PROGRAM Vision_1
VAR
	TON_0: TON;
	Always_ON	:	BOOL	:=TRUE	;//상시 ON
	Always_OFF	:	BOOL	:=FALSE	;//상시 OFF

	

    TON_100MS : TON;
    tPreset_Time : TIME := T#100MS;
	bRun_Timer	:	BOOL	;
	
END_VAR

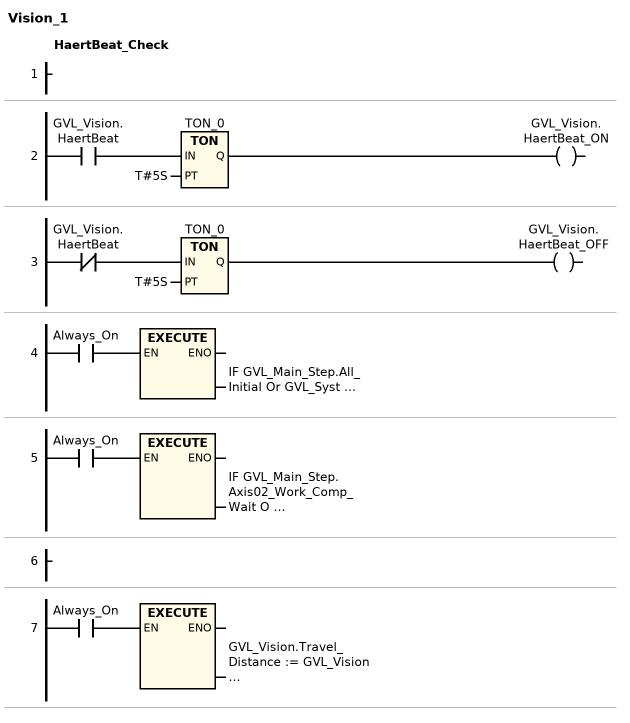
// NETWORK 1: HaertBeat_Check

// NETWORK 2
TON_0(IN := GVL_Vision.HaertBeat, PT := T#5S); // TON
GVL_Vision.HaertBeat_ON := TON_0.Q;

// NETWORK 3
TON_0(IN := NOT GVL_Vision.HaertBeat, PT := T#5S); // TON
GVL_Vision.HaertBeat_OFF := TON_0.Q;

// NETWORK 4
IF Always_On THEN
    IF GVL_Main_Step.All_Initial Or GVL_System.Alarm_Reset THEN
        (* All_Initial이 TRUE일 때, Frame Time을 0으로 초기화 *)
        GVL_Vision.Get_Frame_Time := 0.0;
    END_IF
    bRun_Timer :=GVL_Vision.Vision_Ok AND NOT GVL_Main_Step.Axis04_Work_Comp_Wait;
    TON_100MS(
        IN := bRun_Timer,  
        PT := tPreset_Time,          
        Q  => ,                      
        ET => 
    );
    IF TON_100MS.Q THEN
        
        GVL_Vision.Get_Frame_Time := GVL_Vision.Get_Frame_Time + 0.1;
    	TON_100MS(IN := FALSE);
    
    END_IF
END_IF

// NETWORK 5
IF Always_On THEN
    IF GVL_Main_Step.Axis02_Work_Comp_Wait OR GVL_System.All_Initial THEN
    	GVL_Vision.Data_Read_X	:=	0;
    	GVL_Vision.Data_Read_Y	:=	0;
    	GVL_Vision.Data_Read_R	:=	0;
    	GVL_Vision.Data_Read_X_Vector	:=	0;
    	GVL_Vision.Data_Read_Y_Vector	:=	0;
    	GVL_Vision.Data_Read_R_Vector	:=	0;
    	GVL_Vision.Vision_OK	:=	0;
    	GVL_Vision.Data_Read_OK	:=	0;
    	GVL_Vision.Data_Read_NG	:=	0;
    	GVL_Vision.Get_Frame_Time	:=	0;
    	GVL_Vision.Target_X_Real_Position_Data	:=	0;	
    	GVL_Vision.Press_Speed	:=	0;
    	GVL_Vision.Travel_Distance	:=	0;
    END_IF
END_IF

// NETWORK 6

// NETWORK 7
IF Always_On THEN
    GVL_Vision.Travel_Distance := GVL_Vision.Press_Speed * GVL_Vision.Get_Frame_Time * GVL_Vision.Data_Read_X_Vector;;
    GVL_Vision.Target_X_Real_Position_Data := GVL_Vision.Data_Read_X + GVL_Vision.Travel_Distance;
END_IF

END_PROGRAM

(* stored: Version 1.1.0.1, ProductVersion 3.1.4024.15
   POU Vision_1: Id {81fb605b-be49-42cc-b7e8-bf814d0c125d}, SpecialFunc None *)
